Staubli VAL3: type.pgx

public program type(screen& x_scr, num x_nX, num x_nY, string x_sMessage)
begin
  //-----------------------------------------------------------------------
  //Header begin
  //Description of program
  //  Displays one string to pX column
  //  and pY Line.
  // 显示一个字符串到pX列，pY行。
  //Input parameters
  //  num x_nX :
  //    role : Cursor column
  //    作用：光标列
  //  num x_nY :
  //    role : Cursor row
  //    作用：光标行
  //  string x_sMessage :
  //    role : Message that you want to display
  //   作用：你想去显示的消息
  //Example
  //  call type(scrMy,2,5,"Staubli)
  //
  //History
  //  Creation : 28-04-08 - f.Rob
  //
  //  Modified : 22 Aug 2011 - J. Cook  Added user screens
  //Header end
  //-----------------------------------------------------------------------
  gotoxy(x_scr, x_nX,x_nY)
  put(x_scr, x_sMessage)
end
